PROGRAM MAIN
VAR
END_VAR

END_PROGRAM

(* stored: Version 1.1.0.1
   POU MAIN: Id {77ad10f6-7b8b-4327-8245-e4368394e36d} *)
